Staubli VAL3: checkPoint.pgx

public program checkPoint(bool& x_bCheck[])
begin
  x_bCheck=saveTool:bCheck
end
